FUNCTION_BLOCK ASSEMBLE_AD_FROM_AW (* this Function combines the 2 AW (WORD) adapters to a AD (DWORD) *)
  (* Standard: 61499-2; Description: Copyright (c) 2026 Meisterschulen am Ostbahnhof SPDX-License-Identifier: EPL-2.0 *)
  (* Version 1.0, 2026-05-16, Franz Höpfinger, Meisterschulen am Ostbahnhof, initial API and implementation and/or initial documentation *)
  PACKAGE adapter::assembling;
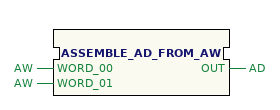
  SOCKETS
    WORD_00 : adapter::types::unidirectional::AW; (* Word 0 *)
    WORD_01 : adapter::types::unidirectional::AW; (* Word 1 *)
  END_SOCKETS
  PLUGS
    OUT : adapter::types::unidirectional::AD; (* DWORD Output *)
  END_PLUGS
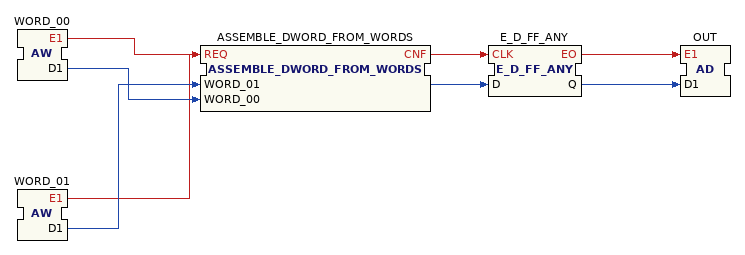
  FBS
    ASSEMBLE_DWORD_FROM_WORDS : eclipse4diac::utils::assembling::ASSEMBLE_DWORD_FROM_WORDS;
    E_D_FF_ANY : iec61499::events::E_D_FF_ANY;
  END_FBS
  EVENT_CONNECTIONS
    WORD_00.E1 TO ASSEMBLE_DWORD_FROM_WORDS.REQ;
    WORD_01.E1 TO ASSEMBLE_DWORD_FROM_WORDS.REQ;
    ASSEMBLE_DWORD_FROM_WORDS.CNF TO E_D_FF_ANY.CLK;
    E_D_FF_ANY.EO TO OUT.E1;
  END_CONNECTIONS
  DATA_CONNECTIONS
    ASSEMBLE_DWORD_FROM_WORDS. TO E_D_FF_ANY.D;
    E_D_FF_ANY.Q TO OUT.D1;
    WORD_01.D1 TO ASSEMBLE_DWORD_FROM_WORDS.WORD_01;
    WORD_00.D1 TO ASSEMBLE_DWORD_FROM_WORDS.WORD_00;
  END_CONNECTIONS
END_FUNCTION_BLOCK
